// Runs executors and active workers assigned to this TwinCAT task.
FUNCTION_BLOCK Thread IMPLEMENTS I_Thread
VAR
	iFirstExecute: _I_Execute;
	iLastExecute: _I_Execute;

	iFirstWorker: I_Worker;
	iLastWorker: I_Worker;

	iPrevThread: I_Thread;
	iNextThread: I_Thread;
END_VAR

PROPERTY INTERNAL _First : _I_Execute
GET
_First := iFirstExecute;
END_GET
END_PROPERTY

PROPERTY INTERNAL _FirstWorker : I_Worker
GET
_FirstWorker := iFirstWorker;
END_GET
END_PROPERTY

PROPERTY INTERNAL _Last : _I_Execute
GET
_Last := iLastExecute;
END_GET
END_PROPERTY

PROPERTY INTERNAL _LastWorker : I_Worker
GET
_LastWorker := iLastWorker;
END_GET
END_PROPERTY

PROPERTY INTERNAL _Next : I_Thread
GET
_Next := iNextThread;
END_GET
SET
iNextThread := _Next;
END_SET
END_PROPERTY

PROPERTY INTERNAL _Prev : I_Thread
GET
_Prev := iPrevThread;
END_GET
SET
iPrevThread := _Prev;
END_SET
END_PROPERTY

METHOD INTERNAL AttachExecute : Result
VAR_INPUT
	iExecute: _I_Execute;
END_VAR
VAR
	iThis: I_Thread := THIS^;
	iThread: I_Thread;
	iPrev: _I_Execute;
	iNext: _I_Execute;
END_VAR
IF iExecute = 0 THEN
	AttachExecute := Error;
	RETURN;
END_IF

iThread := iExecute._Thread;
IF iThread <> iThis THEN
	AttachExecute := Error;
	RETURN;
END_IF

iPrev := iExecute._Prev;
iNext := iExecute._Next;

IF iPrev <> 0 OR iNext <> 0 OR
	iFirstExecute = iExecute OR iLastExecute = iExecute THEN
	Plant.Warn(iExecute, 'Execute attach skipped: execute is already linked in a thread execute list.');
	AttachExecute := None;
    RETURN;
END_IF

iExecute._Prev := iLastExecute;
iExecute._Next := 0;

IF iLastExecute <> 0 THEN
	iLastExecute._Next := iExecute;
	iLastExecute := iExecute;
ELSE
	iFirstExecute := iExecute;
	iLastExecute  := iExecute;
END_IF

AttachExecute := Ok;
END_METHOD

METHOD INTERNAL AttachWorker : Result
VAR_INPUT
	iWorker: I_Worker;
END_VAR
VAR
	iThis: I_Thread := THIS^;
	iThread: I_Thread;
	iPrev: I_Worker;
	iNext: I_Worker;
END_VAR
IF iWorker = 0 THEN
	AttachWorker := Error;
	RETURN;
END_IF

iThread := iWorker.Thread;
IF iThread <> iThis THEN
	AttachWorker := Error;
	RETURN;
END_IF

iPrev := iWorker._Prev;
iNext := iWorker._Next;

IF iPrev <> 0 OR iNext <> 0 OR
	iFirstWorker = iWorker OR iLastWorker = iWorker THEN
	Plant.Warn(iWorker, 'Worker attach skipped: worker is already linked in a thread worker list.');
	AttachWorker := None;
    RETURN;
END_IF

iWorker._Prev := iLastWorker;
iWorker._Next := 0;

IF iLastWorker <> 0 THEN
	iLastWorker._Next := iWorker;
	iLastWorker := iWorker;
ELSE
	iFirstWorker := iWorker;
	iLastWorker  := iWorker;
END_IF

AttachWorker := Ok;
END_METHOD

METHOD INTERNAL DetachExecute : Result
VAR_INPUT
	iExecute: _I_Execute;
END_VAR
VAR
	iThis: I_Thread := THIS^;
	iThread: I_Thread;
	iPrev : _I_Execute;
	iNext : _I_Execute;
END_VAR
IF iExecute = 0 THEN
	DetachExecute := Error;
	RETURN;
END_IF

iThread := iExecute._Thread;
IF iThread <> iThis THEN
	DetachExecute := Error;
	RETURN;
END_IF

iPrev := iExecute._Prev;
iNext := iExecute._Next;

IF iPrev <> 0 THEN
    iPrev._Next := iNext;
END_IF

IF iNext <> 0 THEN
    iNext._Prev := iPrev;
END_IF

IF iFirstExecute = iExecute THEN
    iFirstExecute := iNext;
END_IF

IF iLastExecute = iExecute THEN
    iLastExecute := iPrev;
END_IF

iExecute._Prev := 0;
iExecute._Next := 0;

DetachExecute := Ok;
END_METHOD

METHOD INTERNAL DetachWorker : Result
VAR_INPUT
	iWorker: I_Worker;
END_VAR
VAR
	iThis: I_Thread := THIS^;
	iThread: I_Thread;
	iNext: I_Worker;
	iPrev: I_Worker;
END_VAR
IF iWorker = 0 THEN
	DetachWorker := Error;
	RETURN;
END_IF

iThread := iWorker.Thread;
IF iThread <> iThis THEN
	DetachWorker := Error;
	RETURN;
END_IF

iPrev := iWorker._Prev;
iNext := iWorker._Next;

IF iPrev <> 0 THEN
    iPrev._Next := iNext;
END_IF

IF iNext <> 0 THEN
    iNext._Prev := iPrev;
END_IF

IF iFirstWorker = iWorker THEN
    iFirstWorker := iNext;
END_IF

IF iLastWorker = iWorker THEN
    iLastWorker := iPrev;
END_IF

iWorker._Prev := 0;
iWorker._Next := 0;

DetachWorker := Ok;
END_METHOD

{attribute 'hide'}
METHOD FB_Exit : BOOL
VAR_INPUT
	bInCopyCode: BOOL;
END_VAR
VAR
	iThis: I_Thread := THIS^;
	iMainThread: I_Thread := _Plant.MainThread;
	iExecute: _I_Execute;
	iWorker: I_Worker;
END_VAR
IF NOT bInCopyCode THEN
	IF iThis <> iMainThread THEN
		WHILE iFirstExecute <> 0 DO
			iExecute := iFirstExecute;
			iExecute._Thread := iThis;

			IF DetachExecute(iExecute) <> Ok THEN
				Plant.Panic(iExecute, 'Thread exit failed: could not detach execute before moving it to MainThread.');
				EXIT;
			END_IF

			iExecute._Thread := iMainThread;

			IF IsErr(iMainThread.AttachExecute(iExecute)) THEN
				Plant.Panic(iExecute, 'Thread exit failed: could not attach execute to MainThread before detaching thread.');
				EXIT;
			END_IF

			Plant.Warn(iExecute, 'Thread exit transfer: owning thread left scope; moved execute to MainThread.');
		END_WHILE

		WHILE iFirstWorker <> 0 DO
			iWorker := iFirstWorker;
			iWorker._Thread := iThis;

			IF DetachWorker(iWorker) <> Ok THEN
				Plant.Panic(iWorker, 'Thread exit failed: could not detach worker before moving it to MainThread.');
				EXIT;
			END_IF

			iWorker._Thread := iMainThread;

			IF IsErr(iMainThread.AttachWorker(iWorker)) THEN
				Plant.Panic(iWorker, 'Thread exit failed: could not attach worker to MainThread before detaching thread.');
				EXIT;
			END_IF

			Plant.Warn(iWorker, 'Thread exit transfer: owning thread left scope; moved worker to MainThread.');
		END_WHILE
	END_IF

	Plant._DetachThread(THIS^);
END_IF
END_METHOD

{attribute 'hide'}
METHOD FB_Init : BOOL
VAR_INPUT
	bInitRetains: BOOL;
	bInCopyCode: BOOL;
END_VAR
IF bInCopyCode THEN
	RETURN;
END_IF

IF IsErr(Plant._AttachThread(THIS^)) THEN
	Plant.Panic(THIS^, 'Thread initialization failed: could not attach thread to Plant registry.');
END_IF
END_METHOD

// Processes active workers, then cyclic executors; returns during init or panic.
METHOD Run
VAR
	iWorker: I_Worker := iFirstWorker;
	iExecute: _I_Execute := iFirstExecute;
END_VAR
IF Plant.IsInit OR Plant.Panicked THEN
	RETURN;
END_IF

WHILE iWorker <> 0 DO
	iWorker.Process(iNext => iWorker);
END_WHILE

WHILE iExecute <> 0 DO
	iExecute._Exe(iNext => iExecute);
END_WHILE
END_METHOD

{attribute 'hide'}
METHOD ValidateInterface
VAR_INPUT
END_VAR
END_METHOD

METHOD INTERNAL ValidateThread : Result
VAR CONSTANT
	GUARD: UDINT := Param.VALIDATION_GUARD;
END_VAR
VAR
	iThis: I_Thread := THIS^;
	iExecute: _I_Execute;
	iPrevExecute: _I_Execute;
	iNextExecute: _I_Execute;
	iExecuteThread: I_Thread;
	iWorker: I_Worker;
	iPrevWorker: I_Worker;
	iNextWorker: I_Worker;
	iWorkerThread: I_Thread;
	iCheckExecute: _I_Execute;
	iCheckWorker: I_Worker;
	nGuard: UDINT;
	_err: __SYSTEM.ExceptionCode;
END_VAR
ValidateThread := Error;

__TRY
	IF iFirstExecute = 0 THEN
		IF iLastExecute <> 0 THEN
			Plant.Panic(THIS^, 'Thread validation failed: first execute is 0 but last execute is not 0.');
			RETURN;
		END_IF
	ELSE
		IF Plant.ValidateInterface(iFirstExecute) <> Ok THEN
			Plant.Panic(THIS^, 'Thread validation failed: first execute did not pass ValidateInterface.');
			RETURN;
		END_IF

		IF iLastExecute = 0 THEN
			Plant.Panic(THIS^, 'Thread validation failed: first execute is not 0 but last execute is 0.');
			RETURN;
		END_IF

		IF Plant.ValidateInterface(iLastExecute) <> Ok THEN
			Plant.Panic(THIS^, 'Thread validation failed: last execute did not pass ValidateInterface.');
			RETURN;
		END_IF

		iCheckExecute := iFirstExecute._Prev;
		IF iCheckExecute <> 0 THEN
			Plant.Panic(iFirstExecute, 'Thread validation failed: first execute has a nonzero _Prev link.');
			RETURN;
		END_IF

		iCheckExecute := iLastExecute._Next;
		IF iCheckExecute <> 0 THEN
			Plant.Panic(iLastExecute, 'Thread validation failed: last execute has a nonzero _Next link.');
			RETURN;
		END_IF
	END_IF

	iExecute := iFirstExecute;
	iPrevExecute := 0;
	nGuard := 0;

	WHILE iExecute <> 0 DO
		nGuard := nGuard + 1;
		IF nGuard > GUARD THEN
			Plant.Panic(THIS^, 'Thread validation failed: execute traversal exceeded GUARD; probable cycle.');
			RETURN;
		END_IF

		IF Plant.ValidateInterface(iExecute) <> Ok THEN
			Plant.Panic(THIS^, 'Thread validation failed: current execute did not pass ValidateInterface before link access.');
			RETURN;
		END_IF

		iCheckExecute := iExecute._Prev;
		IF iCheckExecute <> iPrevExecute THEN
			Plant.Panic(iExecute, 'Thread validation failed: current execute _Prev does not match previous visited execute.');
			RETURN;
		END_IF

		iExecuteThread := iExecute._Thread;
		IF Plant.ValidateInterface(iExecuteThread) <> Ok THEN
			Plant.Panic(iExecute, 'Thread validation failed: current execute _Thread is 0 or failed ValidateInterface.');
			RETURN;
		END_IF

		IF iExecuteThread <> iThis THEN
			Plant.Panic(iExecute, 'Thread validation failed: current execute _Thread does not point to the owning thread.');
			RETURN;
		END_IF

		iNextExecute := iExecute._Next;

		IF iNextExecute <> 0 THEN
			IF Plant.ValidateInterface(iNextExecute) <> Ok THEN
				Plant.Panic(iExecute, 'Thread validation failed: current execute _Next did not pass ValidateInterface.');
				RETURN;
			END_IF

			IF iNextExecute = iExecute THEN
				Plant.Panic(iExecute, 'Thread validation failed: current execute _Next points to itself.');
				RETURN;
			END_IF

			iCheckExecute := iNextExecute._Prev;
			IF iCheckExecute <> iExecute THEN
				Plant.Panic(iExecute, 'Thread validation failed: next execute _Prev does not point back to current execute.');
				RETURN;
			END_IF
		END_IF

		iPrevExecute := iExecute;
		iExecute := iNextExecute;
	END_WHILE

	IF iPrevExecute <> iLastExecute THEN
		Plant.Panic(THIS^, 'Thread validation failed: last visited execute does not match thread last execute.');
		RETURN;
	END_IF

	IF iFirstWorker = 0 THEN
		IF iLastWorker <> 0 THEN
			Plant.Panic(THIS^, 'Thread validation failed: first worker is 0 but last worker is not 0.');
			RETURN;
		END_IF
	ELSE
		IF Plant.ValidateInterface(iFirstWorker) <> Ok THEN
			Plant.Panic(THIS^, 'Thread validation failed: first worker did not pass ValidateInterface.');
			RETURN;
		END_IF

		IF iLastWorker = 0 THEN
			Plant.Panic(THIS^, 'Thread validation failed: first worker is not 0 but last worker is 0.');
			RETURN;
		END_IF

		IF Plant.ValidateInterface(iLastWorker) <> Ok THEN
			Plant.Panic(THIS^, 'Thread validation failed: last worker did not pass ValidateInterface.');
			RETURN;
		END_IF

		iCheckWorker := iFirstWorker._Prev;
		IF iCheckWorker <> 0 THEN
			Plant.Panic(iFirstWorker, 'Thread validation failed: first worker has a nonzero _Prev link.');
			RETURN;
		END_IF

		iCheckWorker := iLastWorker._Next;
		IF iCheckWorker <> 0 THEN
			Plant.Panic(iLastWorker, 'Thread validation failed: last worker has a nonzero _Next link.');
			RETURN;
		END_IF
	END_IF

	iWorker := iFirstWorker;
	iPrevWorker := 0;
	nGuard := 0;

	WHILE iWorker <> 0 DO
		nGuard := nGuard + 1;
		IF nGuard > GUARD THEN
			Plant.Panic(THIS^, 'Thread validation failed: worker traversal exceeded GUARD; probable cycle.');
			RETURN;
		END_IF

		IF Plant.ValidateInterface(iWorker) <> Ok THEN
			Plant.Panic(THIS^, 'Thread validation failed: current worker did not pass ValidateInterface before link access.');
			RETURN;
		END_IF

		iCheckWorker := iWorker._Prev;
		IF iCheckWorker <> iPrevWorker THEN
			Plant.Panic(iWorker, 'Thread validation failed: current worker _Prev does not match previous visited worker.');
			RETURN;
		END_IF

		iWorkerThread := iWorker.Thread;
		IF Plant.ValidateInterface(iWorkerThread) <> Ok THEN
			Plant.Panic(iWorker, 'Thread validation failed: current worker Thread is 0 or failed ValidateInterface.');
			RETURN;
		END_IF

		IF iWorkerThread <> iThis THEN
			Plant.Panic(iWorker, 'Thread validation failed: current worker Thread does not point to the owning thread.');
			RETURN;
		END_IF

		iNextWorker := iWorker._Next;

		IF iNextWorker <> 0 THEN
			IF Plant.ValidateInterface(iNextWorker) <> Ok THEN
				Plant.Panic(iWorker, 'Thread validation failed: current worker _Next did not pass ValidateInterface.');
				RETURN;
			END_IF

			IF iNextWorker = iWorker THEN
				Plant.Panic(iWorker, 'Thread validation failed: current worker _Next points to itself.');
				RETURN;
			END_IF

			iCheckWorker := iNextWorker._Prev;
			IF iCheckWorker <> iWorker THEN
				Plant.Panic(iWorker, 'Thread validation failed: next worker _Prev does not point back to current worker.');
				RETURN;
			END_IF
		END_IF

		iPrevWorker := iWorker;
		iWorker := iNextWorker;
	END_WHILE

	IF iPrevWorker <> iLastWorker THEN
		Plant.Panic(THIS^, 'Thread validation failed: last visited worker does not match thread last worker.');
		RETURN;
	END_IF

	ValidateThread := Ok;

__CATCH(_err)
	Plant.Panic(THIS^, 'Thread validation failed: exception while reading validation interfaces or links.');
	ValidateThread := Error;
__ENDTRY
END_METHOD

END_FUNCTION_BLOCK

(* stored: Version 1.1.0.1
   POU Thread: Id {8b3646af-7c89-4248-ba4b-bde043ef6a9a}, SpecialFunc None
   Property _First: Id {a69258e8-ab03-4532-98f4-c6f1e77b0eed}
   Get Get: Id {4db61099-868c-4b8b-90f5-5f62a620bc26}
   Property _FirstWorker: Id {1dc05f76-d766-410c-8416-941e0e2be422}
   Get Get: Id {8662ad19-2a97-4204-a6f0-8b5870da79e2}
   Property _Last: Id {52f96cb0-8ef8-4118-8fe1-42a84f366889}
   Get Get: Id {c5976106-93c4-4bbe-b041-e16625b4868f}
   Property _LastWorker: Id {bbf5e346-34e5-4ec0-8d6a-c990faf1f869}
   Get Get: Id {6cd3e676-9441-416b-b06b-9d8f03331d8b}
   Property _Next: Id {f7a79220-0600-4d7d-9569-b60306c08184}
   Get Get: Id {5d15dfc1-f2fe-46e9-a9a6-648aa0ebd419}
   Set Set: Id {01bf9bf3-7d2b-44de-bd62-73170ec092f1}
   Property _Prev: Id {9f34c22e-ddc3-49b3-9f00-0c3c3179331e}
   Get Get: Id {3740d4ec-b7dc-4312-8675-bf53f4c9ca75}
   Set Set: Id {1f36793c-248f-45df-b3e3-4058cbd74f40}
   Method AttachExecute: Id {09cc9772-526f-41a4-9b80-35664d45d756}
   Method AttachWorker: Id {2efb670a-ea30-4a61-9482-c1d80aa85772}
   Method DetachExecute: Id {2bdcfa7d-9071-4893-8a31-241b3d5383c5}
   Method DetachWorker: Id {186741ed-6fbb-4ec7-ab81-3027a9546f00}
   Method FB_Exit: Id {4d742ca3-01ee-406f-a81f-33459eaeb372}
   Method FB_Init: Id {55119d5d-9bd5-4d72-a24a-603c9384b8f6}
   Method Run: Id {312d03b0-5785-4da7-8eb1-55c23394ad73}
   Method ValidateInterface: Id {c25915fa-ff5e-40d2-928c-da91ae08f4b2}
   Method ValidateThread: Id {a44e3ef3-37a9-495a-b289-edc5f0c924d0} *)
